// TIA Portal project "Mixer" (V19)

(* hardware
DEVICE "S7-1200 station_1"  S7-1200 Station
   slot 0: "Rack_0"  S7-1200 Rack  Rack  V1.0
   slot 1: "PLC_1"  CPU 1212C AC/DC/Rly  6ES7 212-1BE40-0XB0  V4.5
*)

// ===== PLC "PLC_1"  CPU 1212C AC/DC/Rly =====

VAR_GLOBAL   // PLC tag table "Default tag table"
   "FLIPFLOP" AT %M0.0 : Bool;
   "FLIPFLOP2" AT %M0.1 : Bool;
END_VAR

VAR_GLOBAL   // PLC tag table "InputTable"
   "L_LEVEL" AT %I0.0 : Bool;
   "H_LEVEL" AT %I0.1 : Bool;
   "STOP" AT %I0.2 : Bool;
END_VAR

VAR_GLOBAL   // PLC tag table "OutputTable"
   "PUMP_1" AT %Q4.0 : Bool;
   "PUMP_2" AT %Q4.1 : Bool;
   "MIXER" AT %Q4.2 : Bool;
   "VALVE" AT %Q4.3 : Bool;
END_VAR

// folder: System blocks/Program resources

DATA_BLOCK "IEC_Timer_0_DB_1"   // DB2
{ S7_Optimized_Access := 'TRUE' }
AUTHOR : Simatic
FAMILY : IEC
NAME : IEC_TMR
VERSION : 1.0
// stored: InstanceOfName IEC_TIMER
"IEC_TIMER"
BEGIN
END_DATA_BLOCK

// folder: (top level)

ORGANIZATION_BLOCK "Main"   // OB1, LAD, ProgramCycle
TITLE = "Main Program Sweep (Cycle)"
{ S7_Optimized_Access := 'TRUE' }
AUTHOR : Artur Paciorkowski
VERSION : 0.1
   VAR_INPUT
      Initial_Call : Bool;   // Initial call of this OB
      Remanence : Bool;   // =True, if remanent data are available
   END_VAR
BEGIN

REGION Network 1
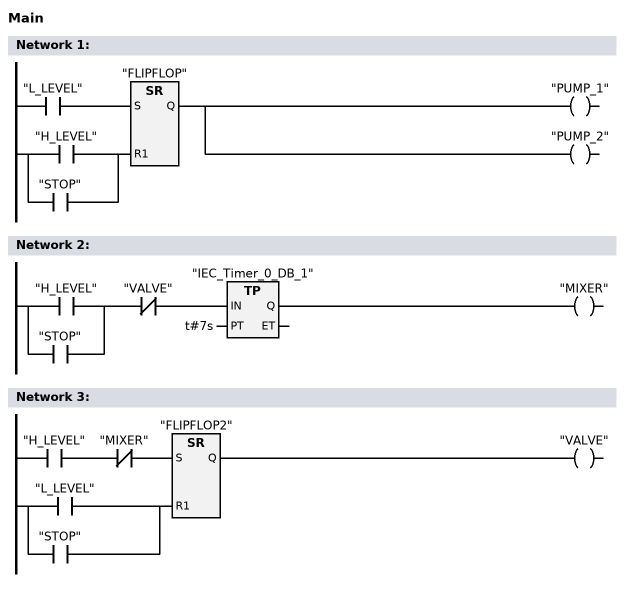
   RUNG wire#powerrail
      Contact( "L_LEVEL" )
      S_SR(operand := "FLIPFLOP", r1 := wire#w1)
      wire#w2
      Coil( "PUMP_1" )
   END_RUNG
   RUNG wire#powerrail
      Contact( "H_LEVEL" )
   END_RUNG wire#w1
   RUNG wire#powerrail
      Contact( "STOP" )
   END_RUNG wire#w1
   RUNG wire#w2
      Coil( "PUMP_2" )
   END_RUNG
   // the same network as SCL:
   IF "L_LEVEL" THEN
       "FLIPFLOP" := TRUE;   // SR flip-flop
   END_IF;
   IF "H_LEVEL" OR "STOP" THEN "FLIPFLOP" := FALSE; END_IF;
   "PUMP_1" := "FLIPFLOP";
   "PUMP_2" := "FLIPFLOP";
END_REGION

REGION Network 2
   "IEC_Timer_0_DB_1".TP(IN := ("H_LEVEL" OR "STOP") AND NOT "VALVE", PT := t#7s);
   "MIXER" := "IEC_Timer_0_DB_1".Q;
END_REGION

REGION Network 3
   RUNG wire#powerrail
      Contact( "H_LEVEL" )
      I_Contact( "MIXER" )
      S_SR(operand := "FLIPFLOP2", r1 := wire#w1)
      Coil( "VALVE" )
   END_RUNG
   RUNG wire#powerrail
      Contact( "L_LEVEL" )
   END_RUNG wire#w1
   RUNG wire#powerrail
      Contact( "STOP" )
   END_RUNG wire#w1
   // the same network as SCL:
   IF "H_LEVEL" AND NOT "MIXER" THEN
       "FLIPFLOP2" := TRUE;   // SR flip-flop
   END_IF;
   IF "L_LEVEL" OR "STOP" THEN "FLIPFLOP2" := FALSE; END_IF;
   "VALVE" := "FLIPFLOP2";
END_REGION
END_ORGANIZATION_BLOCK